TYPE InputBase_8311D824 :
STRUCT
END_STRUCT
END_TYPE

(* stored: Version 1.2.0.0
   DUT InputBase_8311D824: Id {28d1c488-509d-4108-ab68-2bae689168b6} *)
